// TIA Portal project "FactoryIO_Template_S7-1200_V16_V16" (V16)
// Vorlageprojekt für das Buch mit Zielsystem S7-1200

(* hardware
DEVICE "S7-1200-Station_1"  S7-1200 Station
   slot 0: "Baugruppenträger_0"  Rack  V1.0
   slot 1: "PLC_1"  CPU 1211C DC/DC/DC  6ES7 211-1AE40-0XB0  V4.1
*)

// ===== PLC "PLC_1"  CPU 1211C DC/DC/DC =====

VAR_GLOBAL   // PLC tag table "Standard-Variablentabelle"
   "curved conveyor" AT %A0.0 : Bool;
   "start" AT %E0.0 : Bool;
   "stop" AT %E0.1 : Bool;
   "Tag_4" AT %I10.0 : Bool;
   "Tag_5" AT %Q10.0 : Bool;
   "Tag_6" AT %I10.1 : Bool;
   "difuse sensor 1" AT %I0.2 : Bool;
   "difuse sensor 2" AT %I0.3 : Bool;
   "difuse sensor 3" AT %I0.4 : Bool;
   "difuse sensor 4" AT %I0.5 : Bool;
   "difuse sensor 5" AT %I0.6 : Bool;
   "grip detect" AT %I0.7 : Bool;
   "X-moving detect" AT %I1.0 : Bool;
   "Z-moving detect" AT %I1.1 : Bool;
   "conveyor 4" AT %Q0.1 : Bool;
   "conveyor 6" AT %Q0.2 : Bool;
   "X-move" AT %Q0.3 : Bool;
   "Z-move" AT %Q0.4 : Bool;
   "Grip" AT %Q0.5 : Bool;
   "loop marker" AT %M0.0 : Bool;
   "small-box-cond" AT %M0.1 : Bool;
   "Tag_1" AT %M1.0 : Bool;
   "Tag_2" AT %M1.1 : Bool;
   "Tag_3" AT %M0.2 : Bool;
   "z-move-s1" AT %M0.3 : Bool;
   "z-move-s2" AT %M0.4 : Bool;
END_VAR

FUNCTION "MHJ-PLC-Lab-Function-S71200" : Void   // FC9000, SCL
{ S7_Optimized_Access := 'TRUE' }
VERSION : 0.1
   VAR_TEMP
      rdTimeReturn : Int;
      outputTime : DTL;
      SyncVal : Byte;
      forVal : Int;
      forVal_2 : Int;
      Value : Byte;
   END_VAR
   VAR CONSTANT
      CompVal : Byte := 16#34;
      Value_01 : Byte := 16#11;
      Value_01_DW : DWord := 16#A165_D992;
      Value_02_DW : DWord := 16#58BE_4401;
   END_VAR
BEGIN

   #Value:=PEEK(area := 16#82,
        dbNumber := 0,
        byteOffset := 511);
   #Value := #Value + 1;

   POKE(area := 16#82,
        dbNumber := 0,
        byteOffset := 511,
        value := #Value);

   POKE(area:=16#81,
        dbNumber:=0,
        byteOffset:=1016,
        value:=#Value_01_DW);
   POKE(area := 16#81,
        dbNumber := 0,
        byteOffset := 1020,
        value := #Value_02_DW);

   POKE(area := 16#81,
        dbNumber := 0,
        byteOffset := 511,
        value := B#16#00);

   FOR #forVal := 0 TO 120 DO
       FOR #forVal_2:=0 TO 10 DO
           #rdTimeReturn:=RD_SYS_T(#outputTime);
           #rdTimeReturn := WR_SYS_T(#outputTime);
           #rdTimeReturn := RD_SYS_T(#outputTime);
           #rdTimeReturn := WR_SYS_T(#outputTime);
       END_FOR;
       #SyncVal:= PEEK(area := 16#81,
                      dbNumber := 0,
                      byteOffset := 511);
       IF #SyncVal = #CompVal THEN
          GOTO M_1;
       END_IF;
   END_FOR;
   RETURN;

   M_1:
   POKE(area := 16#81,
        dbNumber := 0,
        byteOffset := 511,
        value := B#16#0);
END_FUNCTION

ORGANIZATION_BLOCK "Main"   // OB1, LAD, ProgramCycle
TITLE = "Main Program Sweep (Cycle)"
{ S7_Optimized_Access := 'TRUE' }
VERSION : 0.1
   VAR_INPUT
      Initial_Call : Bool;   // Initial call of this OB
      Remanence : Bool;   // =True, if remanent data are available
   END_VAR
   VAR_TEMP   // added for the SCL form of the ladder/FBD networks
      _w1 : Bool;
   END_VAR
BEGIN

REGION Network 1: Konnektierungsbaustein für PLC-Lab
   // Im Netzwerk 1 wird der Konnektierungsbaustein für PLC-Lab aufgerufen.
   // Dieser Aufruf darf nicht entfernt werden!
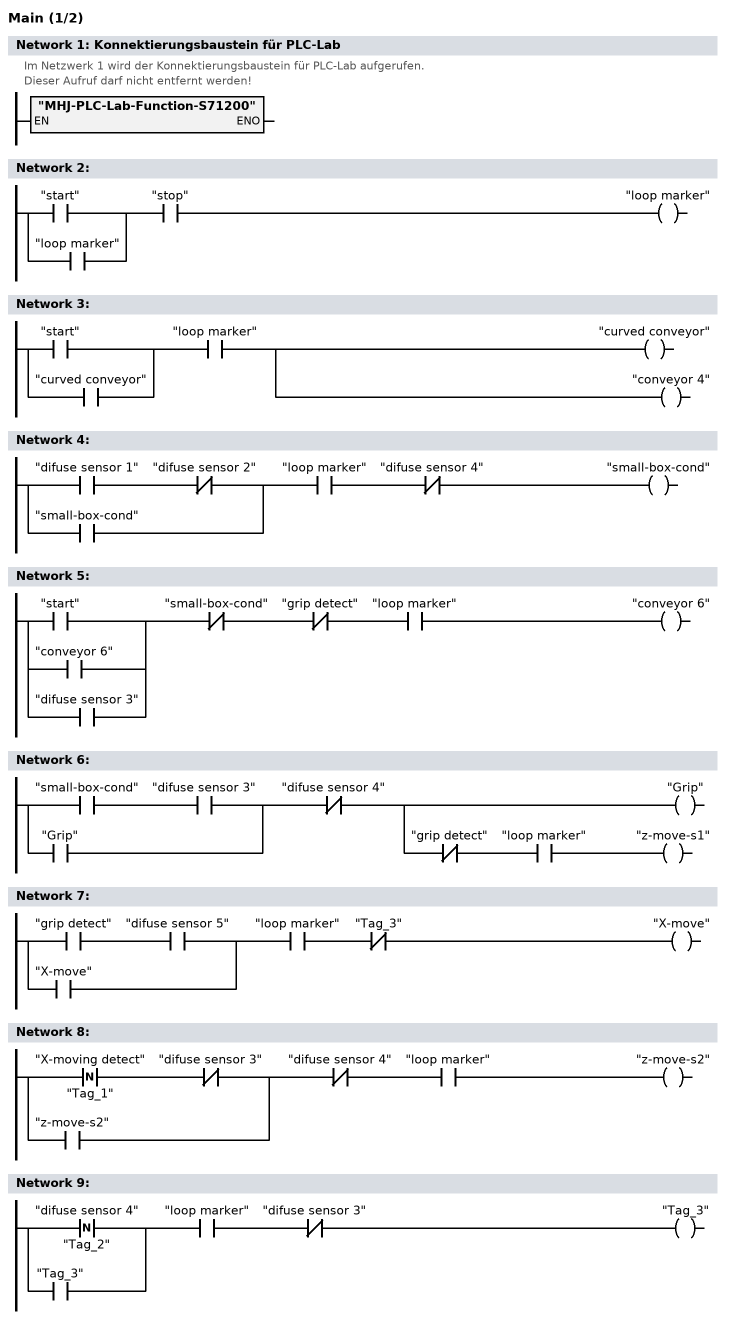
   RUNG wire#powerrail
      "MHJ-PLC-Lab-Function-S71200"()
   END_RUNG
   // the same network as SCL:
   "MHJ-PLC-Lab-Function-S71200"();
END_REGION

REGION Network 2
   RUNG wire#powerrail
      Contact( "start" )
      wire#w1
      Contact( "stop" )
      Coil( "loop marker" )
   END_RUNG
   RUNG wire#powerrail
      Contact( "loop marker" )
   END_RUNG wire#w1
   // the same network as SCL:
   "loop marker" := ("start" OR "loop marker") AND "stop";
END_REGION

REGION Network 3
   RUNG wire#powerrail
      Contact( "start" )
      wire#w1
      Contact( "loop marker" )
      wire#w2
      Coil( "curved conveyor" )
   END_RUNG
   RUNG wire#powerrail
      Contact( "curved conveyor" )
   END_RUNG wire#w1
   RUNG wire#w2
      Coil( "conveyor 4" )
   END_RUNG
   // the same network as SCL:
   "curved conveyor" := ("start" OR "curved conveyor") AND "loop marker";
   "conveyor 4" := "curved conveyor";
END_REGION

REGION Network 4
   RUNG wire#powerrail
      Contact( "difuse sensor 1" )
      I_Contact( "difuse sensor 2" )
      wire#w1
      Contact( "loop marker" )
      I_Contact( "difuse sensor 4" )
      Coil( "small-box-cond" )
   END_RUNG
   RUNG wire#powerrail
      Contact( "small-box-cond" )
   END_RUNG wire#w1
   // the same network as SCL:
   "small-box-cond" := (("difuse sensor 1" AND NOT "difuse sensor 2") OR "small-box-cond") AND "loop marker" AND NOT "difuse sensor 4";
END_REGION

REGION Network 5
   RUNG wire#powerrail
      Contact( "start" )
      wire#w1
      I_Contact( "small-box-cond" )
      I_Contact( "grip detect" )
      Contact( "loop marker" )
      Coil( "conveyor 6" )
   END_RUNG
   RUNG wire#powerrail
      Contact( "conveyor 6" )
   END_RUNG wire#w1
   RUNG wire#powerrail
      Contact( "difuse sensor 3" )
   END_RUNG wire#w1
   // the same network as SCL:
   "conveyor 6" := ("start" OR "conveyor 6" OR "difuse sensor 3") AND NOT "small-box-cond" AND NOT "grip detect" AND "loop marker";
END_REGION

REGION Network 6
   RUNG wire#powerrail
      Contact( "small-box-cond" )
      Contact( "difuse sensor 3" )
      wire#w1
      I_Contact( "difuse sensor 4" )
      wire#w2
      Coil( "Grip" )
   END_RUNG
   RUNG wire#powerrail
      Contact( "Grip" )
   END_RUNG wire#w1
   RUNG wire#w2
      I_Contact( "grip detect" )
      Contact( "loop marker" )
      Coil( "z-move-s1" )
   END_RUNG
   // the same network as SCL:
   "Grip" := (("small-box-cond" AND "difuse sensor 3") OR "Grip") AND NOT "difuse sensor 4";
   "z-move-s1" := "Grip" AND NOT "grip detect" AND "loop marker";
END_REGION

REGION Network 7
   RUNG wire#powerrail
      Contact( "grip detect" )
      Contact( "difuse sensor 5" )
      wire#w1
      Contact( "loop marker" )
      I_Contact( "Tag_3" )
      Coil( "X-move" )
   END_RUNG
   RUNG wire#powerrail
      Contact( "X-move" )
   END_RUNG wire#w1
   // the same network as SCL:
   "X-move" := (("grip detect" AND "difuse sensor 5") OR "X-move") AND "loop marker" AND NOT "Tag_3";
END_REGION

REGION Network 8
   RUNG wire#powerrail
      N_Contact(operand := "X-moving detect", bit := "Tag_1")
      I_Contact( "difuse sensor 3" )
      wire#w1
      I_Contact( "difuse sensor 4" )
      Contact( "loop marker" )
      Coil( "z-move-s2" )
   END_RUNG
   RUNG wire#powerrail
      Contact( "z-move-s2" )
   END_RUNG wire#w1
   // the same network as SCL:
   #_w1 := NOT "X-moving detect" AND "Tag_1";   // falling edge of "X-moving detect"
   "Tag_1" := "X-moving detect";
   "z-move-s2" := ((#_w1 AND NOT "difuse sensor 3") OR "z-move-s2") AND NOT "difuse sensor 4" AND "loop marker";
END_REGION

REGION Network 9
   RUNG wire#powerrail
      N_Contact(operand := "difuse sensor 4", bit := "Tag_2")
      wire#w1
      Contact( "loop marker" )
      I_Contact( "difuse sensor 3" )
      Coil( "Tag_3" )
   END_RUNG
   RUNG wire#powerrail
      Contact( "Tag_3" )
   END_RUNG wire#w1
   // the same network as SCL:
   #_w1 := NOT "difuse sensor 4" AND "Tag_2";   // falling edge of "difuse sensor 4"
   "Tag_2" := "difuse sensor 4";
   "Tag_3" := (#_w1 OR "Tag_3") AND "loop marker" AND NOT "difuse sensor 3";
END_REGION

REGION Network 10
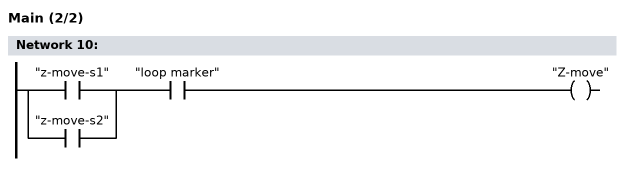
   RUNG wire#powerrail
      Contact( "z-move-s1" )
      wire#w1
      Contact( "loop marker" )
      Coil( "Z-move" )
   END_RUNG
   RUNG wire#powerrail
      Contact( "z-move-s2" )
   END_RUNG wire#w1
   // the same network as SCL:
   "Z-move" := ("z-move-s1" OR "z-move-s2") AND "loop marker";
END_REGION
END_ORGANIZATION_BLOCK